PROGRAM MAIN2
VAR
	btn			:BOOL;
	btnStart	: BOOL;
	btnStop 	: BOOL := TRUE;
	Coil: BOOL;
	
END_VAR

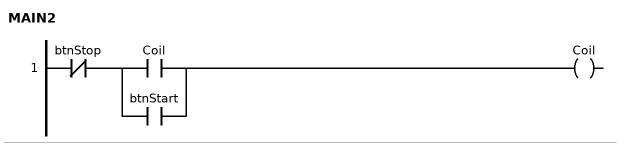
// NETWORK 1
Coil := NOT btnStop AND (Coil OR btnStart);

END_PROGRAM

(* stored: Version 1.1.0.1, ProductVersion 3.1.4024.6
   POU MAIN2: Id {171c6829-d940-48da-97fc-a8de090dbc26}, SpecialFunc None *)
